PROGRAM MAIN
VAR
	{attribute 'OPC.UA.DA' := '1'}
	state: XY_Stage_State; (* XY Stage State *)
	
	// motor variables
	axisX		: AXIS_REF;
	axisY		: AXIS_REF;
	fbXReset	: MC_Reset;
	fbYReset	: MC_Reset;
	fbXPower	: MC_Power;
	fbYPower	: MC_Power;
	fbXMoveAbs	: MC_MoveAbsolute;
	fbYMoveAbs	: MC_MoveAbsolute;
	bReset		: BOOL := FALSE;
	bXEnable	: BOOL := FALSE;
	bYEnable	: BOOL := FALSE;
	bMove		: BOOL := FALSE;
	fXTargetPos	: LREAL := 0;
	fYTargetPos : LREAL := 0;
	fXTargetVel : LREAL := 360;
	fYTargetVel : LREAL := 360;
	
	// inputs
	{attribute 'OPC.UA.DA' := '1'}
	inputXPos	: LREAL := 0;
	{attribute 'OPC.UA.DA' := '1'}
	inputYPos	: LREAL := 0;
	{attribute 'OPC.UA.DA' := '1'}
	inputXVel	: LREAL := 360;
	{attribute 'OPC.UA.DA' := '1'}
	inputYVel	: LREAL := 360;
	
	// outputs
	{attribute 'OPC.UA.DA' := '1'}
	{attribute 'OPC.UA.DA.Access' := '1'}
	XPos		: LREAL; (* X position *)
	{attribute 'OPC.UA.DA' := '1'}
	{attribute 'OPC.UA.DA.Access' := '1'}
	YPos		: LREAL; (* Y position *)
	{attribute 'OPC.UA.DA' := '1'}
	{attribute 'OPC.UA.DA.Access' := '1'}
	XVel		: LREAL; (* X velocity *)
	{attribute 'OPC.UA.DA' := '1'}
	{attribute 'OPC.UA.DA.Access' := '1'}
	YVel		: LREAL; (* Y velocity *)
	{attribute 'OPC.UA.DA' := '1'}
	{attribute 'OPC.UA.DA.Access' := '1'}
	XLag		: LREAL := 0; (* X position lag *)
	{attribute 'OPC.UA.DA' := '1'}
	{attribute 'OPC.UA.DA.Access' := '1'}
	YLag		: LREAL := 0; (* Y position lag *)
	{attribute 'OPC.UA.DA' := '1'}
	{attribute 'OPC.UA.DA.Access' := '1'}
	XLagMax		: LREAL := 0; (* maximum X position lag (abs val) *)
	{attribute 'OPC.UA.DA' := '1'}
	{attribute 'OPC.UA.DA.Access' := '1'}
	YLagMax		: LREAL := 0; (* maximum Y position lag (abs val) *)
	{attribute 'OPC.UA.DA' := '1'}
	{attribute 'OPC.UA.DA.Access' := '1'}
	XErrorCode		: UDINT := 0; (* last error code for X *)
	{attribute 'OPC.UA.DA' := '1'}
	{attribute 'OPC.UA.DA.Access' := '1'}
	YErrorCode		: UDINT := 0; (* last error code for Y *)
	
END_VAR

axisX.ReadStatus();
axisY.ReadStatus();

// process input & output variables
// these limits taken from Drive Manager
inputXVel := MIN(inputXVel, 6744);
inputYVel := MIN(inputYVel, 6744);

XPos := axisX.NcToPlc.ActPos;
YPos := axisY.NcToPlc.ActPos;
XVel := axisX.NcToPlc.ActVelo;
YVel := axisY.NcToPlc.ActVelo;
XLag := axisX.NcToPlc.PosDiff;
YLag := axisY.NcToPlc.PosDiff;
XLagMax := MAX(ABS(XLag), XLagMax);
YLagMax := MAX(ABS(YLag), YLagMax);

IF axisX.Status.Error = TRUE OR axisY.Status.Error = TRUE OR
	fbXPower.Error = TRUE OR fbYPower.Error = TRUE OR
	fbXMoveAbs.Error = TRUE OR fbYMoveAbs.Error = TRUE THEN
	XErrorCode := MAX(axisX.Status.ErrorID, fbXPower.ErrorID, fbXMoveAbs.ErrorID);
	YErrorCode := MAX(axisY.Status.ErrorID, fbYPower.ErrorID, fbYMoveAbs.ErrorID);
	state := XY_Stage_State.error;
END_IF

CASE state OF
XY_Stage_State.off: // init (power off)
	bReset := FALSE;
	bXEnable := FALSE;
	bYEnable := FALSE;
	bMove := FALSE;
XY_Stage_State.reset: // reset & enable power to axes
	bReset := TRUE;
	bXEnable := FALSE; // FIX temporary
	bYEnable := TRUE;
	XErrorCode := 0;
	YErrorCode := 0;
	IF fbXReset.Done = TRUE AND fbYReset.Done = TRUE AND
		// FIX fbXPower.Status = TRUE AND fbYPower.Status = TRUE THEN
		fbYPower.Status = TRUE THEN
		bReset := FALSE;
		state := XY_Stage_State.ready;
	END_IF
XY_Stage_State.ready: // set up move
	fXTargetPos := inputXPos;
	fYTargetPos := inputYPos;
	fXTargetVel := inputXVel;
	fYTargetVel := inputYVel;
	bMove := TRUE;
	state := XY_Stage_State.moving;
XY_Stage_State.moving: // moving
	// FIX IF fbXMoveAbs.Done = TRUE AND fbYMoveAbs.Done = TRUE THEN
	IF fbYMoveAbs.Done = TRUE THEN
		bMove := FALSE;
		state := XY_Stage_State.ready;
	END_IF
XY_Stage_State.error: // error
	RETURN; // lock into this state
END_CASE

// function blocks, execution controlled by their execute bits
fbXReset(Axis := axisX, Execute := bReset);
fbYReset(Axis := axisY, Execute := bReset);

fbXPower(
	Axis := axisX,
	Enable := bXEnable,
	Enable_Positive := bXEnable,
	Enable_Negative := bXEnable,
	Override := 100);
fbYPower(
	Axis := axisY,
	Enable := bYEnable,
	Enable_Positive := bYEnable,
	Enable_Negative := bYEnable,
	Override := 100);
	
fbXMoveAbs(
	Axis:= axisX,
	Execute:= bMove,
	Position:= fXTargetPos,
	Velocity:= fXTargetVel,
	Acceleration:= ,
	Deceleration:= ,
	Jerk:= );
fbYMoveAbs(
	Axis:= axisY,
	Execute:= bMove,
	Position:= fYTargetPos,
	Velocity:= fYTargetVel,
	Acceleration:= ,
	Deceleration:= ,
	Jerk:= );

END_PROGRAM

(* stored: Version 1.1.0.1, ProductVersion 3.1.4024.6
   POU MAIN: Id {0d52fe34-3379-4937-8bfa-de5557a85529}, SpecialFunc None *)
